SUBAPPLICATION logiBUS_IXA_BG_OPC_AX (* logiBUS DI Kanal: VT-Hintergrundfarbe + OPC-UA-Publish (generisch, ein Kanal) *)
  (* Standard: 61499-2; Description: Copyright (c) 2023 Meisterschulen am Ostbahnhof This program and the accompanying materials are made available under the terms of the Eclipse Public License 2.0 which is available at https://www.eclipse.org/legal/epl-2.0/ SPDX-License-Identifier: EPL-2.0 *)
  (* Version 1.0, 2023-10-23, Franz Höpfinger, Meisterschulen am Ostbahnhof, initial API and implementation and/or initial documentation *)
  PACKAGE MyLib_AX::sys;
  IMPORT isobus::UT::Q::const::IDs::ID_NULL;
  IMPORT logiBUS::io::DI::logiBUS_DI;
  IMPORT logiBUS::io::DI::logiBUS_DI_S;
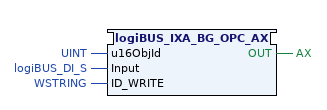
  VAR_INPUT
    u16ObjId : UINT := ID_NULL; (* Object ID Hintergrund-Rechteck (VT), ID_NULL = noch kein VT-Objekt *)
    Input : logiBUS::io::DI::logiBUS_DI_S := logiBUS_DI::Invalid; (* Identify the Input Input_I1..I8 *)
    ID_WRITE : WSTRING; (* OPC-UA Publish-Key (lesbar) *)
  END_VAR
  PLUGS
    OUT : adapter::types::unidirectional::AX;
  END_PLUGS
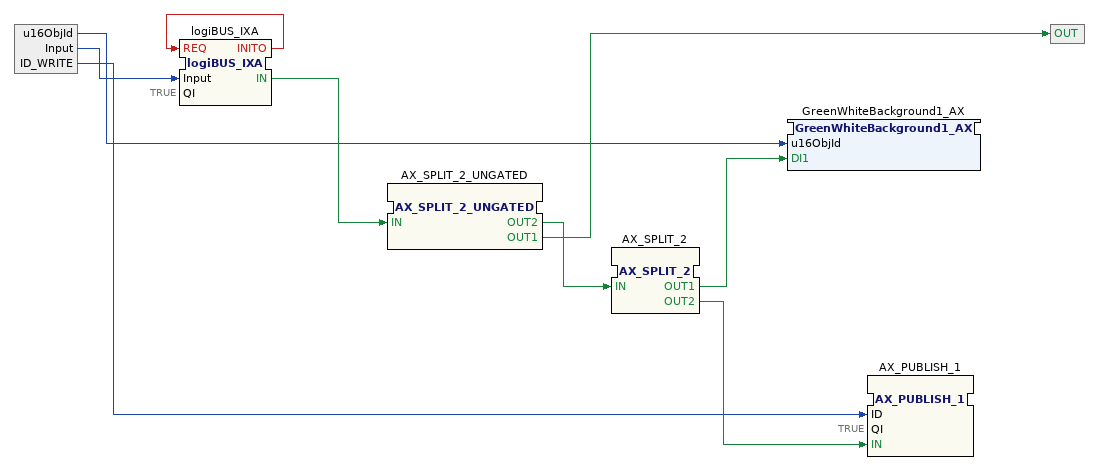
  FBS
    logiBUS_IXA : logiBUS::io::DI::logiBUS_IXA(QI := TRUE);
    AX_PUBLISH_1 : adapter::net::AX_PUBLISH_1(QI := TRUE);
    AX_SPLIT_2 : adapter::events::unidirectional::AX_SPLIT_2;
    AX_SPLIT_2_UNGATED : adapter::events::unidirectional::AX_SPLIT_2_UNGATED;
  END_FBS
  SUBAPPS
    GreenWhiteBackground1_AX : MyLib::sys::GreenWhiteBackground1_AX;
  END_SUBAPPS
  EVENT_CONNECTIONS
    logiBUS_IXA.INITO TO logiBUS_IXA.REQ;
  END_CONNECTIONS
  DATA_CONNECTIONS
    Input TO logiBUS_IXA.Input;
    u16ObjId TO GreenWhiteBackground1_AX.u16ObjId;
    ID_WRITE TO AX_PUBLISH_1.ID;
  END_CONNECTIONS
  ADAPTER_CONNECTIONS
    logiBUS_IXA.IN TO AX_SPLIT_2_UNGATED.IN;
    AX_SPLIT_2.OUT1 TO GreenWhiteBackground1_AX.DI1;
    AX_SPLIT_2.OUT2 TO AX_PUBLISH_1.IN;
    AX_SPLIT_2_UNGATED.OUT2 TO AX_SPLIT_2.IN;
    AX_SPLIT_2_UNGATED.OUT1 TO OUT;
  END_CONNECTIONS
END_SUBAPPLICATION
